{attribute wpf [Container(Layout.Stack)]}
TYPE StackLayout:
STRUCT
	_wheel: Wheel;
END_STRUCT
END_TYPE

(* stored: Version 1.1.0.1, ProductVersion 3.1.4024.9
   DUT StackLayout: Id {1be459b3-4f78-4c87-bebf-5f3b887461ed} *)
